Universal Robots PolyScope program: move_down_test.urp

Program move_down_test (installation=default directory=/programs/Tests createdIn=5.9.1.1031110 lastSavedIn=5.9.1.1031110 robotSerialNumber=20185500256)
Calibrated DH parameters: a=[0.000163, -0.146131, -0.38577, 0.000126, -0.000021, 0]; d=[0.161954, 188.306531, -157.478086, -30.695088, 0.099716, 0.099628]; alpha=[1.569701, -0.00212, 0.002263, 1.570438, -1.570123, 0]; deltaTheta=[0, -1.219859, 7.681919, -0.178877, -0.000001, 0]
Robot Program (runOnlyOnce=true)
  MoveJ speed 60 deg/s, acceleration 80 deg/s^2 (useActiveTCP=true) feature=Base
    Waypoint Waypoint (Variable): variable(featureName=cam_bin1)
  MoveJ speed 60 deg/s, acceleration 80 deg/s^2 (useActiveTCP=true) feature=Base
    Waypoint Waypoint (Variable): variable(featureName=above_bin1)
  Call MoveDownUntilContact
SubProgram -> MoveDownUntilContact
SubProgram MoveDownUntilContact (keepSynchronizedWithDisk=false)
  MoveL speed 250 mm/s, acceleration 1200 mm/s^2 (useActiveTCP=true) feature=Base
    MoveDirectionNode (selectedDirection=ZMinus toolParams=0.05, 0.3) feature(featureName=base_plate)
      Until TOOL_CONTACT_DETECTION (allowActions=false retraction=0.005 decelerationAcceleration=1 decelerationAngularAcceleration=34.906585)
